TYPE ST_PneumaticAxisConfig :
STRUCT
    bSafetyShutter: BOOL := FALSE; //Bit to define if pneumatic axis is Shutter needing PSS permit
    sPneumaticAxisName: String(32);
    nTimeLimitMovingWithValveOn: INT; //User defined time limit for moving with valve on in seconds
    nTimeLimitMovingWithValveOff: INT; //User defined time limit for moving with valve off in seconds
    eSelectPneumaticAxisGroup: E_PneumaticAxisGroup; //Select the pneumatic group 1 or 2, to connect to the correct pressure sensor
	ePneumaticAxisMode: E_PneumaticAxisMode := E_PneumaticAxisMode.eMonostable;
END_STRUCT
END_TYPE

(* stored: Version 1.1.0.1
   DUT ST_PneumaticAxisConfig: Id {f7d3b15a-c25b-0a63-3175-d55d3daa4326} *)
